PROGRAM MAIN
VAR
	MyDword		: DWORD;
	ScannerIndex	: UINT;
	
	bitResult		: BOOL;
END_VAR


bitResult	:= F_ReturnBitInDword(inDword:= MyDword,inIndex:= ScannerIndex);

END_PROGRAM

(* stored: Version 1.1.0.1, ProductVersion 3.1.4024.12
   POU MAIN: Id {b0072296-03da-449f-b748-a2297b045a0f}, SpecialFunc None *)
